// TIA Portal V17 export
// export: Created 2025-08-05T09:35:57.6788297Z, ExportSetting WithDefaults, DisplayName Totally Integrated Automation Portal, DisplayVersion V17, DisplayName TIA Portal Openness, DisplayVersion V17, DisplayName TIA Portal Version Control Interface, DisplayVersion V17, DisplayName SINAMICS Startdrive Advanced, DisplayVersion V17, DisplayName SINAMICS Startdrive G130, G150, S120, S150, SINAMICS MV, S210, DisplayVersion V17, DisplayName SINAMICS Startdrive G110M, G120, G120C, G120D, G120P, G115D, DisplayVersion V17, DisplayName STEP 7 Professional, DisplayVersion V17, DisplayName STEP 7 Safety, DisplayVersion V17, DisplayName WinCC Advanced, DisplayVersion V17
FUNCTION_BLOCK "IPG_Weld_Interface"   // FB304, LAD
TITLE = IPG Communication Handling / IPG Weld Interface
{ S7_Optimized_Access := 'FALSE' }
VERSION : 1.0
// stored: AutoNumber true, IsIECCheckEnabled false, SetENOAutomatically false, UDAEnableTagReadback false
   VAR_INPUT
      iScanner : "Scanner_Inputs";
      iYLS : "YLS_Inputs";
      iInstance_Index : Int;
      iYLR_Power_On : Bool;
      bYLR : Bool;
      bYLS : Bool;
   END_VAR
   VAR_OUTPUT
      oScanner : "Scanner_Outputs";
      oYLS : "YLS_Outputs";
      oYLR_Laser_On : Bool;
      oYLR_Reset : Bool;
   END_VAR
   VAR DB_SPECIFIC
      sStep : Int;
      sLast_Step : Int;
      sScanner_Idle : Bool;
      sScanner_Active : Bool;
      sScanner_Error : Bool;
      sScanner_Waiting_Enable : Bool;
      sScanner_Waiting_Strobe : Bool;
      sScanner_Waiting_Start : Bool;
      tJob_Start_ONS { ExternalAccessible := 'False'; ExternalVisible := 'False'; ExternalWritable := 'False'} : Bool;
      tJob_Stop_ONS { ExternalAccessible := 'False'; ExternalVisible := 'False'; ExternalWritable := 'False'} : Bool;
      siScanner_Job : Byte;
      siScanner_Group : Byte;
      soScanner_Job : Byte;
      soScanner_Group : Byte;
      sVersion { S7_SetPoint := 'True'} : Real;
      sStepTimeout : IEC_TIMER;
      sReset_Timer { S7_SetPoint := 'True'} : IEC_TIMER;
      sLog : Array[0..50] of Struct
         Load_Start_Time : Date_And_Time;
         Load_Stop_Time : Date_And_Time;
         Fire_Start_Time : Date_And_Time;
         Fire_Stop_Time : Date_And_Time;
         Job_ID : Byte;
         Group_ID : Byte;
      END_STRUCT;
      sBlankLog : Struct
         Load_Start_Time : Date_And_Time;
         Load_Stop_Time : Date_And_Time;
         Fire_Start_Time : Date_And_Time;
         Fire_Stop_Time : Date_And_Time;
         Job_ID : Byte;
         Group_ID : Byte;
      END_STRUCT;
   END_VAR
   VAR_TEMP
      tLasRes : Bool;
      tStep_Changed_ONS : Bool;
      tPointer : Int;
      tStart_Load_Int : Int;
      tStop_Load_Int : Int;
      tStart_Fire_Int : Int;
      tStop_Fire_Int : Int;
   END_VAR
   VAR_TEMP   // added for the SCL form of the ladder/FBD networks
      _w1 : Bool;
      _w2 : Bool;
   END_VAR
BEGIN

REGION Network 1: Version
   // V1.1
   // Mapped all Scanner and YLS Inputs and Outputs
   // V1.2
   // Added YLR Faults and Interface (need to add condition for Power On of YLR)
   // V2
   // Laser Comm DB Reorder, remove redunudant logic
   // Added Job and Group Log
   // Removed Guide Beam On Fault. Soace reserved.
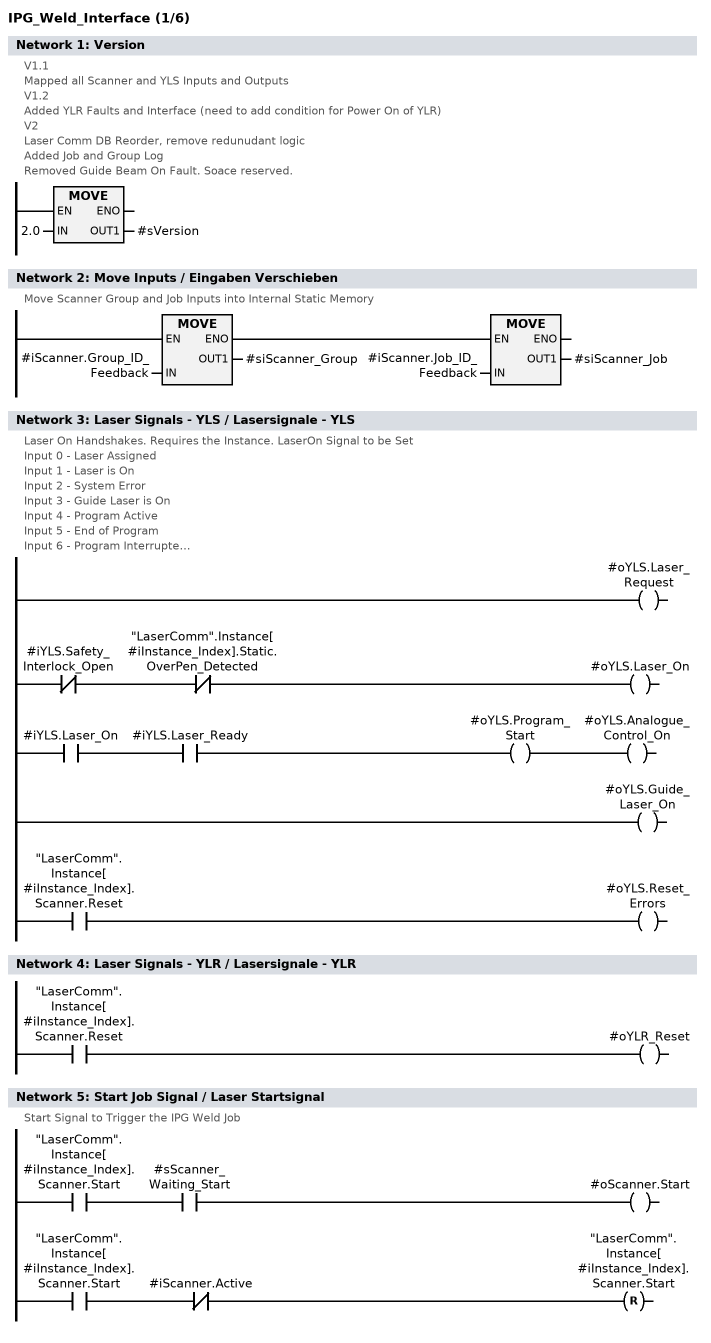
   RUNG wire#powerrail
      Move(in := 2.0, out1 => #sVersion)
   END_RUNG
   // the same network as SCL:
   #sVersion := 2.0;
END_REGION

REGION Network 2: Move Inputs / Eingaben Verschieben
   // Move Scanner Group and Job Inputs into Internal Static Memory
   RUNG wire#powerrail
      Move(in := #iScanner.Group_ID_Feedback, out1 => #siScanner_Group)
      Move(in := #iScanner.Job_ID_Feedback, out1 => #siScanner_Job)
   END_RUNG
   // the same network as SCL:
   #siScanner_Group := #iScanner.Group_ID_Feedback;
   #siScanner_Job := #iScanner.Job_ID_Feedback;
END_REGION

REGION Network 3: Laser Signals - YLS / Lasersignale - YLS
   // Laser On Handshakes. Requires the Instance. LaserOn Signal to be Set
   // Input 0 - Laser Assigned
   // Input 1 - Laser is On
   // Input 2 - System Error
   // Input 3 - Guide Laser is On
   // Input 4 - Program Active
   // Input 5 - End of Program
   // Input 6 - Program Interrupted
   // Input 7 - Analogue Control is On
   // Input 8 - System Warning
   // Input 9 - Laser Ready
   // Input 10 - Emission On
   // 
   // Output 0 - Laser Request (should always be On)
   // Output 1 - Laser On
   // Output 2 - Reset Errors
   // Output 3 - Guide Laser On
   // Output 4 - Program Start
   // Output 5 - Program Stop
   // Output 6 - Reserved
   // Output 7 - Analogue Control On
   RUNG wire#powerrail
      Coil( #oYLS.Laser_Request )
   END_RUNG
   RUNG wire#powerrail
      I_Contact( #iYLS.Safety_Interlock_Open )
      I_Contact( "LaserComm".Instance[#iInstance_Index].Static.OverPen_Detected )
      Coil( #oYLS.Laser_On )
   END_RUNG
   RUNG wire#powerrail
      Contact( #iYLS.Laser_On )
      Contact( #iYLS.Laser_Ready )
      Coil( #oYLS.Program_Start )
      Coil( #oYLS.Analogue_Control_On )
   END_RUNG
   RUNG wire#powerrail
      Coil( #oYLS.Guide_Laser_On )
   END_RUNG
   RUNG wire#powerrail
      Contact( "LaserComm".Instance[#iInstance_Index].Scanner.Reset )
      Coil( #oYLS.Reset_Errors )
   END_RUNG
   // the same network as SCL:
   #oYLS.Laser_Request := TRUE;
   #oYLS.Laser_On := NOT #iYLS.Safety_Interlock_Open AND NOT "LaserComm".Instance[#iInstance_Index].Static.OverPen_Detected;
   #oYLS.Program_Start := #iYLS.Laser_On AND #iYLS.Laser_Ready;
   #oYLS.Analogue_Control_On := #oYLS.Program_Start;
   #oYLS.Guide_Laser_On := TRUE;
   #oYLS.Reset_Errors := "LaserComm".Instance[#iInstance_Index].Scanner.Reset;
END_REGION

REGION Network 4: Laser Signals - YLR / Lasersignale - YLR
   RUNG wire#powerrail
      Contact( "LaserComm".Instance[#iInstance_Index].Scanner.Reset )
      Coil( #oYLR_Reset )
   END_RUNG
   // the same network as SCL:
   #oYLR_Reset := "LaserComm".Instance[#iInstance_Index].Scanner.Reset;
END_REGION

REGION Network 5: Start Job Signal / Laser Startsignal
   // Start Signal to Trigger the IPG Weld Job
   RUNG wire#powerrail
      Contact( "LaserComm".Instance[#iInstance_Index].Scanner.Start )
      Contact( #sScanner_Waiting_Start )
      Coil( #oScanner.Start )
   END_RUNG
   RUNG wire#powerrail
      Contact( "LaserComm".Instance[#iInstance_Index].Scanner.Start )
      I_Contact( #iScanner.Active )
      R_Coil( "LaserComm".Instance[#iInstance_Index].Scanner.Start )
   END_RUNG
   // the same network as SCL:
   #oScanner.Start := "LaserComm".Instance[#iInstance_Index].Scanner.Start AND #sScanner_Waiting_Start;
   IF "LaserComm".Instance[#iInstance_Index].Scanner.Start AND NOT #iScanner.Active THEN
       "LaserComm".Instance[#iInstance_Index].Scanner.Start := FALSE;
   END_IF;
END_REGION

REGION Network 6: Log Fire Time Handling
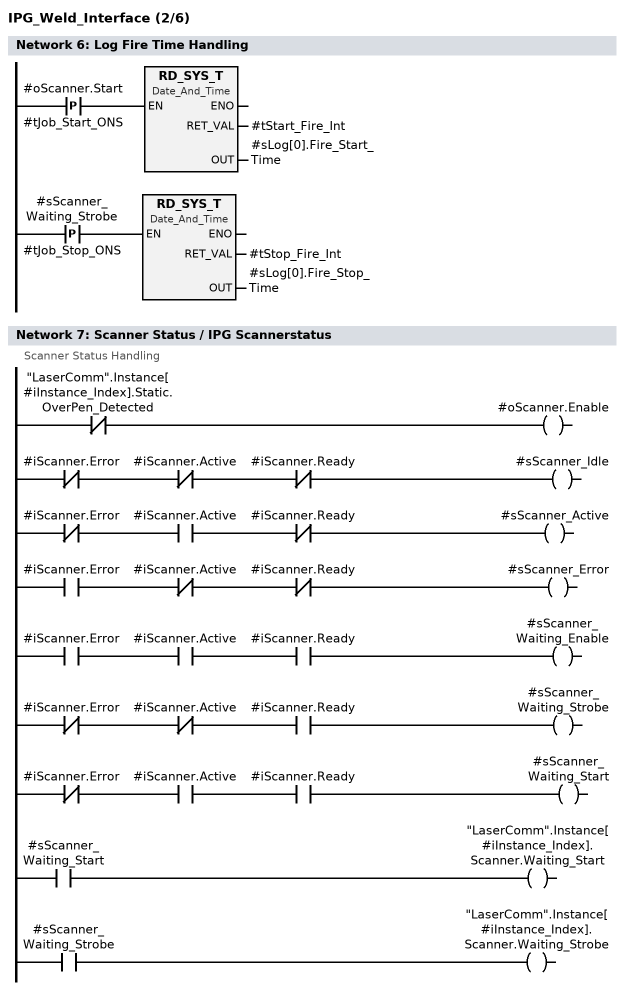
   RUNG wire#powerrail
      P_Contact(operand := #oScanner.Start, bit := #tJob_Start_ONS)
      { S7_Templates := "date_type := Date_And_Time" } RD_SYS_T(RET_VAL => #tStart_Fire_Int, OUT => #sLog[0].Fire_Start_Time)
   END_RUNG
   RUNG wire#powerrail
      P_Contact(operand := #sScanner_Waiting_Strobe, bit := #tJob_Stop_ONS)
      { S7_Templates := "date_type := Date_And_Time" } RD_SYS_T(RET_VAL => #tStop_Fire_Int, OUT => #sLog[0].Fire_Stop_Time)
   END_RUNG
   // the same network as SCL:
   #_w1 := #oScanner.Start AND NOT #tJob_Start_ONS;   // rising edge of #oScanner.Start
   #tJob_Start_ONS := #oScanner.Start;
   IF #_w1 THEN #tStart_Fire_Int := RD_SYS_T(OUT => #sLog[0].Fire_Start_Time); END_IF;
   #_w2 := #sScanner_Waiting_Strobe AND NOT #tJob_Stop_ONS;   // rising edge of #sScanner_Waiting_Strobe
   #tJob_Stop_ONS := #sScanner_Waiting_Strobe;
   IF #_w2 THEN #tStop_Fire_Int := RD_SYS_T(OUT => #sLog[0].Fire_Stop_Time); END_IF;
END_REGION

REGION Network 7: Scanner Status / IPG Scannerstatus
   // Scanner Status Handling
   RUNG wire#powerrail
      I_Contact( "LaserComm".Instance[#iInstance_Index].Static.OverPen_Detected )
      Coil( #oScanner.Enable )
   END_RUNG
   RUNG wire#powerrail
      I_Contact( #iScanner.Error )
      I_Contact( #iScanner.Active )
      I_Contact( #iScanner.Ready )
      Coil( #sScanner_Idle )
   END_RUNG
   RUNG wire#powerrail
      I_Contact( #iScanner.Error )
      Contact( #iScanner.Active )
      I_Contact( #iScanner.Ready )
      Coil( #sScanner_Active )
   END_RUNG
   RUNG wire#powerrail
      Contact( #iScanner.Error )
      I_Contact( #iScanner.Active )
      I_Contact( #iScanner.Ready )
      Coil( #sScanner_Error )
   END_RUNG
   RUNG wire#powerrail
      Contact( #iScanner.Error )
      Contact( #iScanner.Active )
      Contact( #iScanner.Ready )
      Coil( #sScanner_Waiting_Enable )
   END_RUNG
   RUNG wire#powerrail
      I_Contact( #iScanner.Error )
      I_Contact( #iScanner.Active )
      Contact( #iScanner.Ready )
      Coil( #sScanner_Waiting_Strobe )
   END_RUNG
   RUNG wire#powerrail
      I_Contact( #iScanner.Error )
      Contact( #iScanner.Active )
      Contact( #iScanner.Ready )
      Coil( #sScanner_Waiting_Start )
   END_RUNG
   RUNG wire#powerrail
      Contact( #sScanner_Waiting_Start )
      Coil( "LaserComm".Instance[#iInstance_Index].Scanner.Waiting_Start )
   END_RUNG
   RUNG wire#powerrail
      Contact( #sScanner_Waiting_Strobe )
      Coil( "LaserComm".Instance[#iInstance_Index].Scanner.Waiting_Strobe )
   END_RUNG
   // the same network as SCL:
   #oScanner.Enable := NOT "LaserComm".Instance[#iInstance_Index].Static.OverPen_Detected;
   #sScanner_Idle := NOT #iScanner.Error AND NOT #iScanner.Active AND NOT #iScanner.Ready;
   #sScanner_Active := NOT #iScanner.Error AND #iScanner.Active AND NOT #iScanner.Ready;
   #sScanner_Error := #iScanner.Error AND NOT #iScanner.Active AND NOT #iScanner.Ready;
   #sScanner_Waiting_Enable := #iScanner.Error AND #iScanner.Active AND #iScanner.Ready;
   #sScanner_Waiting_Strobe := NOT #iScanner.Error AND NOT #iScanner.Active AND #iScanner.Ready;
   #sScanner_Waiting_Start := NOT #iScanner.Error AND #iScanner.Active AND #iScanner.Ready;
   "LaserComm".Instance[#iInstance_Index].Scanner.Waiting_Start := #sScanner_Waiting_Start;
   "LaserComm".Instance[#iInstance_Index].Scanner.Waiting_Strobe := #sScanner_Waiting_Strobe;
END_REGION

REGION Network 8: Step 0 / Schritt 0
   // Initial Step. Wait for Scanner Ready to Begin with Job and Group Not 0. / Job und Gruppen ID Laden
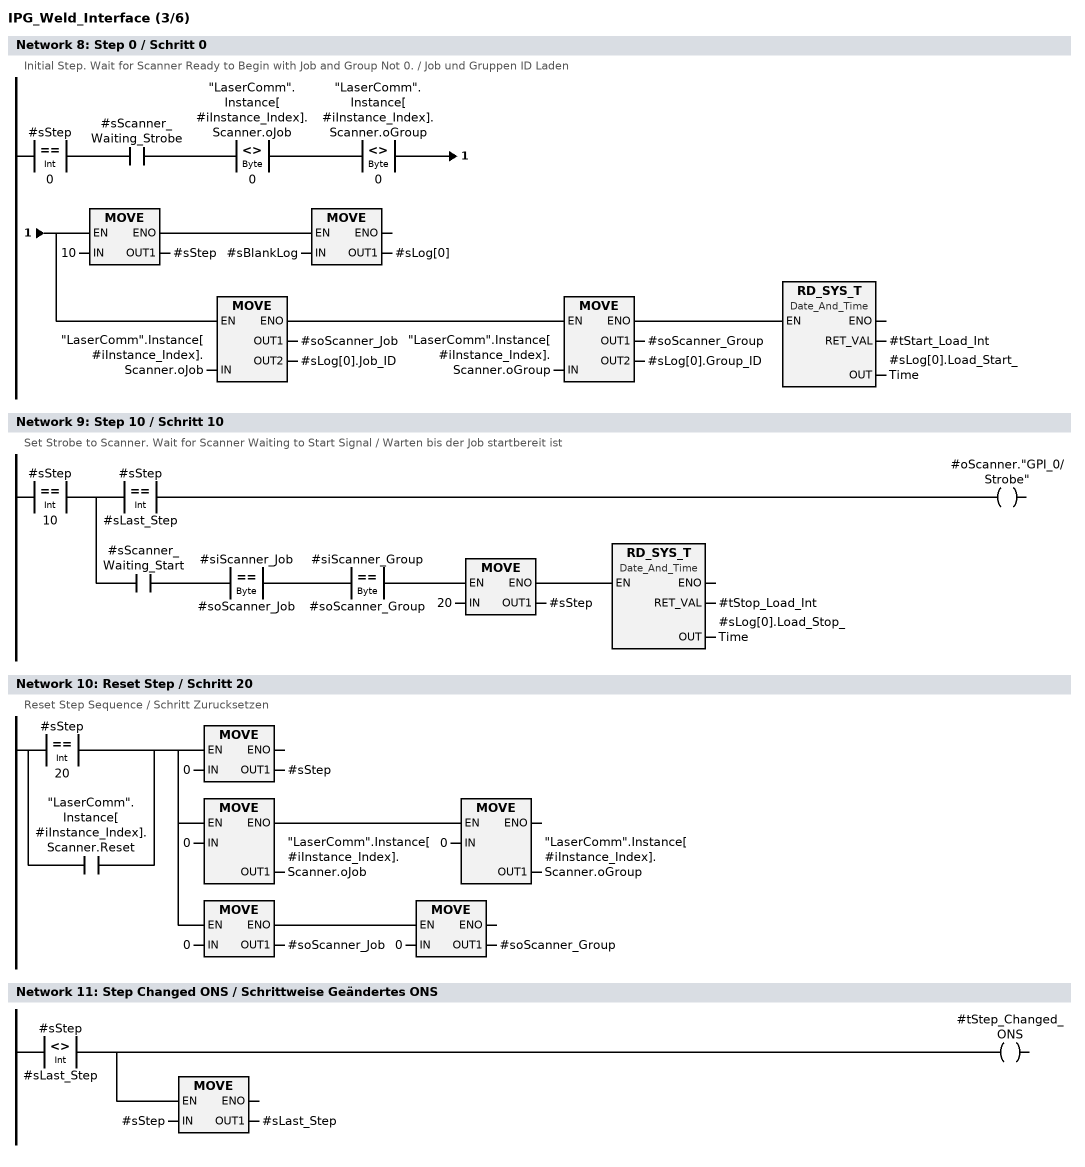
   RUNG wire#powerrail
      { S7_Templates := "SrcType := Int" } EQ_Contact(in1 := #sStep, in2 := 0)
      Contact( #sScanner_Waiting_Strobe )
      { S7_Templates := "SrcType := Byte" } NE_Contact(in1 := "LaserComm".Instance[#iInstance_Index].Scanner.oJob, in2 := 0)
      { S7_Templates := "SrcType := Byte" } NE_Contact(in1 := "LaserComm".Instance[#iInstance_Index].Scanner.oGroup, in2 := 0)
      wire#w1
      Move(in := 10, out1 => #sStep)
      Move(in := #sBlankLog, out1 => #sLog[0])
   END_RUNG
   RUNG wire#w1
      Move(in := "LaserComm".Instance[#iInstance_Index].Scanner.oJob, out1 => #soScanner_Job, out2 => #sLog[0].Job_ID)
      Move(in := "LaserComm".Instance[#iInstance_Index].Scanner.oGroup, out1 => #soScanner_Group, out2 => #sLog[0].Group_ID)
      { S7_Templates := "date_type := Date_And_Time" } RD_SYS_T(RET_VAL => #tStart_Load_Int, OUT => #sLog[0].Load_Start_Time)
   END_RUNG
   // the same network as SCL:
   #_w1 := (#sStep = 0) AND #sScanner_Waiting_Strobe AND ("LaserComm".Instance[#iInstance_Index].Scanner.oJob <> 0) AND ("LaserComm".Instance[#iInstance_Index].Scanner.oGroup <> 0);
   #_w2 := (#sStep = 0) AND #sScanner_Waiting_Strobe AND ("LaserComm".Instance[#iInstance_Index].Scanner.oJob <> 0) AND ("LaserComm".Instance[#iInstance_Index].Scanner.oGroup <> 0);
   IF #_w2 THEN
       #sStep := 10;
       #sLog[0] := #sBlankLog;
   END_IF;
   IF #_w1 THEN
       #soScanner_Job := "LaserComm".Instance[#iInstance_Index].Scanner.oJob;
       #sLog[0].Job_ID := "LaserComm".Instance[#iInstance_Index].Scanner.oJob;
       #soScanner_Group := "LaserComm".Instance[#iInstance_Index].Scanner.oGroup;
       #sLog[0].Group_ID := "LaserComm".Instance[#iInstance_Index].Scanner.oGroup;
       #tStart_Load_Int := RD_SYS_T(OUT => #sLog[0].Load_Start_Time);
   END_IF;
END_REGION

REGION Network 9: Step 10 / Schritt 10
   // Set Strobe to Scanner. Wait for Scanner Waiting to Start Signal / Warten bis der Job startbereit ist
   RUNG wire#powerrail
      { S7_Templates := "SrcType := Int" } EQ_Contact(in1 := #sStep, in2 := 10)
      wire#w1
      { S7_Templates := "SrcType := Int" } EQ_Contact(in1 := #sStep, in2 := #sLast_Step)
      Coil( #oScanner."GPI_0/Strobe" )
   END_RUNG
   RUNG wire#w1
      Contact( #sScanner_Waiting_Start )
      { S7_Templates := "SrcType := Byte" } EQ_Contact(in1 := #siScanner_Job, in2 := #soScanner_Job)
      { S7_Templates := "SrcType := Byte" } EQ_Contact(in1 := #siScanner_Group, in2 := #soScanner_Group)
      Move(in := 20, out1 => #sStep)
      { S7_Templates := "date_type := Date_And_Time" } RD_SYS_T(RET_VAL => #tStop_Load_Int, OUT => #sLog[0].Load_Stop_Time)
   END_RUNG
   // the same network as SCL:
   #_w1 := #sStep = 10;
   #oScanner."GPI_0/Strobe" := #_w1 AND (#sStep = #sLast_Step);
   IF #_w1 AND #sScanner_Waiting_Start AND (#siScanner_Job = #soScanner_Job) AND (#siScanner_Group = #soScanner_Group) THEN
       #sStep := 20;
       #tStop_Load_Int := RD_SYS_T(OUT => #sLog[0].Load_Stop_Time);
   END_IF;
END_REGION

REGION Network 10: Reset Step / Schritt 20
   // Reset Step Sequence / Schritt Zurucksetzen
   RUNG wire#powerrail
      { S7_Templates := "SrcType := Int" } EQ_Contact(in1 := #sStep, in2 := 20)
      wire#w1
      Move(in := 0, out1 => #sStep)
   END_RUNG
   RUNG wire#powerrail
      Contact( "LaserComm".Instance[#iInstance_Index].Scanner.Reset )
   END_RUNG wire#w1
   RUNG wire#w1
      Move(in := 0, out1 => "LaserComm".Instance[#iInstance_Index].Scanner.oJob)
      Move(in := 0, out1 => "LaserComm".Instance[#iInstance_Index].Scanner.oGroup)
   END_RUNG
   RUNG wire#w1
      Move(in := 0, out1 => #soScanner_Job)
      Move(in := 0, out1 => #soScanner_Group)
   END_RUNG
   // the same network as SCL:
   #_w1 := (#sStep = 20) OR "LaserComm".Instance[#iInstance_Index].Scanner.Reset;
   IF #_w1 THEN
       #sStep := 0;
       "LaserComm".Instance[#iInstance_Index].Scanner.oJob := 0;
       "LaserComm".Instance[#iInstance_Index].Scanner.oGroup := 0;
       #soScanner_Job := 0;
       #soScanner_Group := 0;
   END_IF;
END_REGION

REGION Network 11: Step Changed ONS / Schrittweise Geändertes ONS
   RUNG wire#powerrail
      { S7_Templates := "SrcType := Int" } NE_Contact(in1 := #sStep, in2 := #sLast_Step)
      wire#w1
      Coil( #tStep_Changed_ONS )
   END_RUNG
   RUNG wire#w1
      { S7_GenerateENO := "TRUE" } Move(in := #sStep, out1 => #sLast_Step)
   END_RUNG
   // the same network as SCL:
   #tStep_Changed_ONS := #sStep <> #sLast_Step;
   IF #tStep_Changed_ONS THEN #sLast_Step := #sStep; END_IF;
END_REGION

REGION Network 12: Reset Flag / Reset Flag Entrigein
   // Clear Reset Flag - Timer Required as Laser Source requires a duration pulse to reset
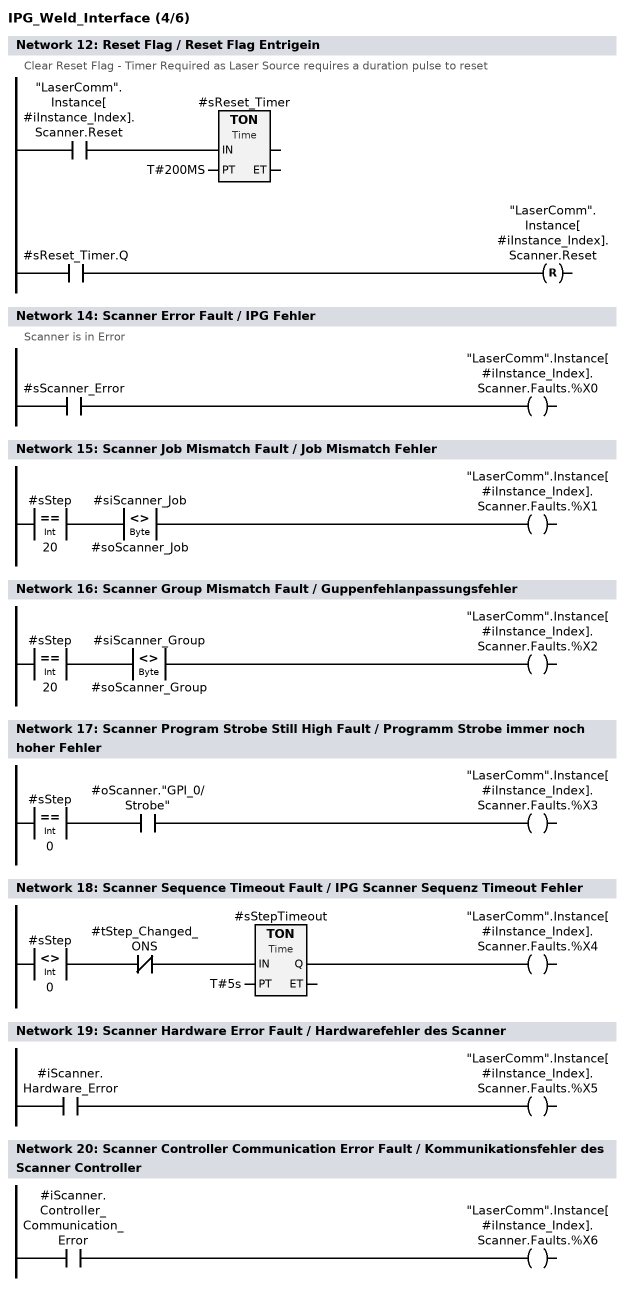
   RUNG wire#powerrail
      Contact( "LaserComm".Instance[#iInstance_Index].Scanner.Reset )
      { S7_Templates := "time_type := Time" } #sReset_Timer.TON(pt := T#200MS, et =>)
   END_RUNG
   RUNG wire#powerrail
      Contact( #sReset_Timer.Q )
      R_Coil( "LaserComm".Instance[#iInstance_Index].Scanner.Reset )
   END_RUNG
   // the same network as SCL:
   #sReset_Timer.TON(IN := "LaserComm".Instance[#iInstance_Index].Scanner.Reset, PT := T#200MS);
   IF #sReset_Timer.Q THEN "LaserComm".Instance[#iInstance_Index].Scanner.Reset := FALSE; END_IF;
END_REGION

REGION Network 13 (SCL): Job Log Handler
   // Records when the last job and group was loaded and fired
   // Job Log Handler

   IF #sLog[0].Job_ID <> 0 AND #sLog[0].Group_ID <> 0 AND #sLog[0].Fire_Stop_Time <> DT#1990-01-01-00:00:00 THEN
       FOR #tPointer := 49 TO 0 BY -1 DO
           #sLog[#tPointer + 1] := #sLog[#tPointer];
       END_FOR;

       #sLog[0] := #sBlankLog;

   END_IF;
END_REGION

REGION Network 14: Scanner Error Fault / IPG Fehler
   // Scanner is in Error
   RUNG wire#powerrail
      Contact( #sScanner_Error )
      Coil( "LaserComm".Instance[#iInstance_Index].Scanner.Faults.%X0 )
   END_RUNG
   // the same network as SCL:
   "LaserComm".Instance[#iInstance_Index].Scanner.Faults.%X0 := #sScanner_Error;
END_REGION

REGION Network 15: Scanner Job Mismatch Fault / Job Mismatch Fehler
   RUNG wire#powerrail
      { S7_Templates := "SrcType := Int" } EQ_Contact(in1 := #sStep, in2 := 20)
      { S7_Templates := "SrcType := Byte" } NE_Contact(in1 := #siScanner_Job, in2 := #soScanner_Job)
      Coil( "LaserComm".Instance[#iInstance_Index].Scanner.Faults.%X1 )
   END_RUNG
   // the same network as SCL:
   "LaserComm".Instance[#iInstance_Index].Scanner.Faults.%X1 := (#sStep = 20) AND (#siScanner_Job <> #soScanner_Job);
END_REGION

REGION Network 16: Scanner Group Mismatch Fault / Guppenfehlanpassungsfehler
   RUNG wire#powerrail
      { S7_Templates := "SrcType := Int" } EQ_Contact(in1 := #sStep, in2 := 20)
      { S7_Templates := "SrcType := Byte" } NE_Contact(in1 := #siScanner_Group, in2 := #soScanner_Group)
      Coil( "LaserComm".Instance[#iInstance_Index].Scanner.Faults.%X2 )
   END_RUNG
   // the same network as SCL:
   "LaserComm".Instance[#iInstance_Index].Scanner.Faults.%X2 := (#sStep = 20) AND (#siScanner_Group <> #soScanner_Group);
END_REGION

REGION Network 17: Scanner Program Strobe Still High Fault / Programm Strobe immer noch hoher Fehler
   RUNG wire#powerrail
      { S7_Templates := "SrcType := Int" } EQ_Contact(in1 := #sStep, in2 := 0)
      Contact( #oScanner."GPI_0/Strobe" )
      Coil( "LaserComm".Instance[#iInstance_Index].Scanner.Faults.%X3 )
   END_RUNG
   // the same network as SCL:
   "LaserComm".Instance[#iInstance_Index].Scanner.Faults.%X3 := (#sStep = 0) AND #oScanner."GPI_0/Strobe";
END_REGION

REGION Network 18: Scanner Sequence Timeout Fault / IPG Scanner Sequenz Timeout Fehler
   RUNG wire#powerrail
      { S7_Templates := "SrcType := Int" } NE_Contact(in1 := #sStep, in2 := 0)
      I_Contact( #tStep_Changed_ONS )
      { S7_Templates := "time_type := Time" } #sStepTimeout.TON(pt := T#5s, et =>)
      Coil( "LaserComm".Instance[#iInstance_Index].Scanner.Faults.%X4 )
   END_RUNG
   // the same network as SCL:
   #sStepTimeout.TON(IN := (#sStep <> 0) AND NOT #tStep_Changed_ONS, PT := T#5s);
   "LaserComm".Instance[#iInstance_Index].Scanner.Faults.%X4 := #sStepTimeout.Q;
END_REGION

REGION Network 19: Scanner Hardware Error Fault / Hardwarefehler des Scanner
   RUNG wire#powerrail
      Contact( #iScanner.Hardware_Error )
      Coil( "LaserComm".Instance[#iInstance_Index].Scanner.Faults.%X5 )
   END_RUNG
   // the same network as SCL:
   "LaserComm".Instance[#iInstance_Index].Scanner.Faults.%X5 := #iScanner.Hardware_Error;
END_REGION

REGION Network 20: Scanner Controller Communication Error Fault / Kommunikationsfehler des Scanner Controller
   RUNG wire#powerrail
      Contact( #iScanner.Controller_Communication_Error )
      Coil( "LaserComm".Instance[#iInstance_Index].Scanner.Faults.%X6 )
   END_RUNG
   // the same network as SCL:
   "LaserComm".Instance[#iInstance_Index].Scanner.Faults.%X6 := #iScanner.Controller_Communication_Error;
END_REGION

REGION Network 21: Scanner Head Communication Error Fault / Fehler bei derKommunikation mit dem Scannerkopf
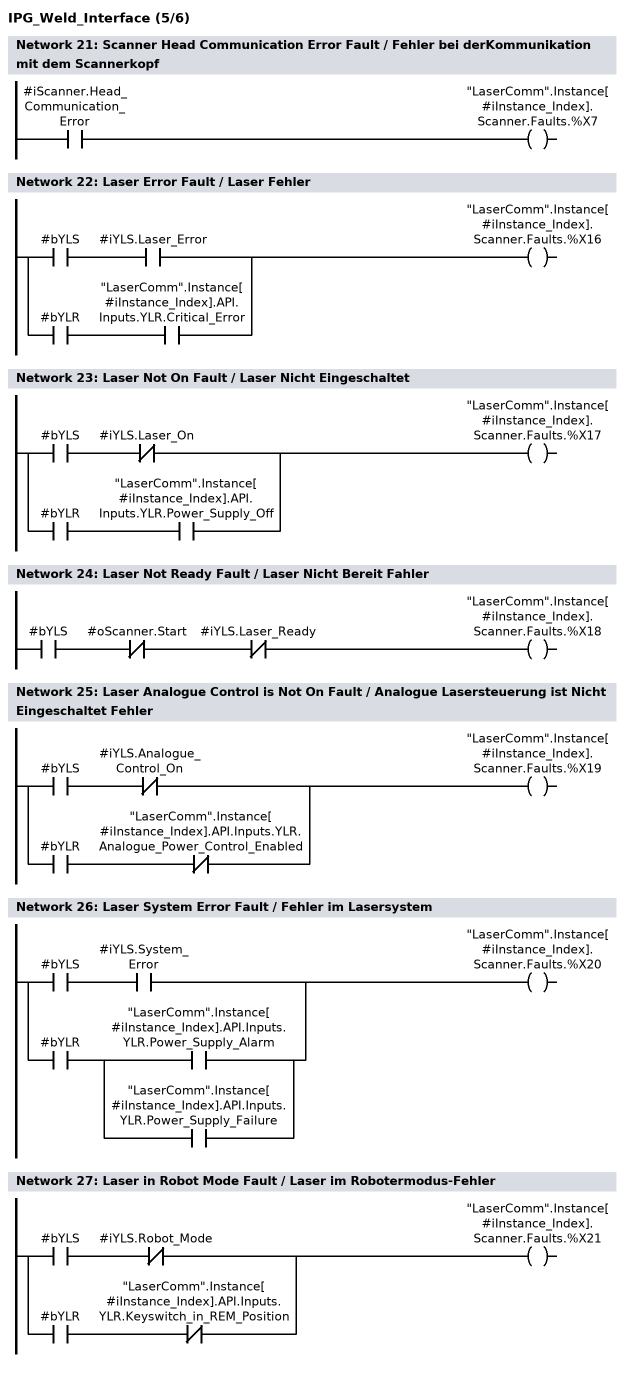
   RUNG wire#powerrail
      Contact( #iScanner.Head_Communication_Error )
      Coil( "LaserComm".Instance[#iInstance_Index].Scanner.Faults.%X7 )
   END_RUNG
   // the same network as SCL:
   "LaserComm".Instance[#iInstance_Index].Scanner.Faults.%X7 := #iScanner.Head_Communication_Error;
END_REGION

REGION Network 22: Laser Error Fault / Laser Fehler
   RUNG wire#powerrail
      Contact( #bYLS )
      Contact( #iYLS.Laser_Error )
      wire#w1
      Coil( "LaserComm".Instance[#iInstance_Index].Scanner.Faults.%X16 )
   END_RUNG
   RUNG wire#powerrail
      Contact( #bYLR )
      Contact( "LaserComm".Instance[#iInstance_Index].API.Inputs.YLR.Critical_Error )
   END_RUNG wire#w1
   // the same network as SCL:
   "LaserComm".Instance[#iInstance_Index].Scanner.Faults.%X16 := (#bYLS AND #iYLS.Laser_Error) OR (#bYLR AND "LaserComm".Instance[#iInstance_Index].API.Inputs.YLR.Critical_Error);
END_REGION

REGION Network 23: Laser Not On Fault / Laser Nicht Eingeschaltet
   RUNG wire#powerrail
      Contact( #bYLS )
      I_Contact( #iYLS.Laser_On )
      wire#w1
      Coil( "LaserComm".Instance[#iInstance_Index].Scanner.Faults.%X17 )
   END_RUNG
   RUNG wire#powerrail
      Contact( #bYLR )
      Contact( "LaserComm".Instance[#iInstance_Index].API.Inputs.YLR.Power_Supply_Off )
   END_RUNG wire#w1
   // the same network as SCL:
   "LaserComm".Instance[#iInstance_Index].Scanner.Faults.%X17 := (#bYLS AND NOT #iYLS.Laser_On) OR (#bYLR AND "LaserComm".Instance[#iInstance_Index].API.Inputs.YLR.Power_Supply_Off);
END_REGION

REGION Network 24: Laser Not Ready Fault / Laser Nicht Bereit Fahler
   RUNG wire#powerrail
      Contact( #bYLS )
      I_Contact( #oScanner.Start )
      I_Contact( #iYLS.Laser_Ready )
      Coil( "LaserComm".Instance[#iInstance_Index].Scanner.Faults.%X18 )
   END_RUNG
   // the same network as SCL:
   "LaserComm".Instance[#iInstance_Index].Scanner.Faults.%X18 := #bYLS AND NOT #oScanner.Start AND NOT #iYLS.Laser_Ready;
END_REGION

REGION Network 25: Laser Analogue Control is Not On Fault / Analogue Lasersteuerung ist Nicht Eingeschaltet Fehler
   RUNG wire#powerrail
      Contact( #bYLS )
      I_Contact( #iYLS.Analogue_Control_On )
      wire#w1
      Coil( "LaserComm".Instance[#iInstance_Index].Scanner.Faults.%X19 )
   END_RUNG
   RUNG wire#powerrail
      Contact( #bYLR )
      I_Contact( "LaserComm".Instance[#iInstance_Index].API.Inputs.YLR.Analogue_Power_Control_Enabled )
   END_RUNG wire#w1
   // the same network as SCL:
   "LaserComm".Instance[#iInstance_Index].Scanner.Faults.%X19 := (#bYLS AND NOT #iYLS.Analogue_Control_On) OR (#bYLR AND NOT "LaserComm".Instance[#iInstance_Index].API.Inputs.YLR.Analogue_Power_Control_Enabled);
END_REGION

REGION Network 26: Laser System Error Fault / Fehler im Lasersystem
   RUNG wire#powerrail
      Contact( #bYLS )
      Contact( #iYLS.System_Error )
      wire#w1
      Coil( "LaserComm".Instance[#iInstance_Index].Scanner.Faults.%X20 )
   END_RUNG
   RUNG wire#powerrail
      Contact( #bYLR )
      wire#w2
      Contact( "LaserComm".Instance[#iInstance_Index].API.Inputs.YLR.Power_Supply_Alarm )
   END_RUNG wire#w1
   RUNG wire#w2
      Contact( "LaserComm".Instance[#iInstance_Index].API.Inputs.YLR.Power_Supply_Failure )
   END_RUNG wire#w1
   // the same network as SCL:
   "LaserComm".Instance[#iInstance_Index].Scanner.Faults.%X20 := (#bYLS AND #iYLS.System_Error) OR (#bYLR AND ("LaserComm".Instance[#iInstance_Index].API.Inputs.YLR.Power_Supply_Alarm OR "LaserComm".Instance[#iInstance_Index].API.Inputs.YLR.Power_Supply_Failure));
END_REGION

REGION Network 27: Laser in Robot Mode Fault / Laser im Robotermodus-Fehler
   RUNG wire#powerrail
      Contact( #bYLS )
      I_Contact( #iYLS.Robot_Mode )
      wire#w1
      Coil( "LaserComm".Instance[#iInstance_Index].Scanner.Faults.%X21 )
   END_RUNG
   RUNG wire#powerrail
      Contact( #bYLR )
      I_Contact( "LaserComm".Instance[#iInstance_Index].API.Inputs.YLR.Keyswitch_in_REM_Position )
   END_RUNG wire#w1
   // the same network as SCL:
   "LaserComm".Instance[#iInstance_Index].Scanner.Faults.%X21 := (#bYLS AND NOT #iYLS.Robot_Mode) OR (#bYLR AND NOT "LaserComm".Instance[#iInstance_Index].API.Inputs.YLR.Keyswitch_in_REM_Position);
END_REGION

REGION Network 28: Laser Interlock Open Fault / Fehler Laserverriegelung offen
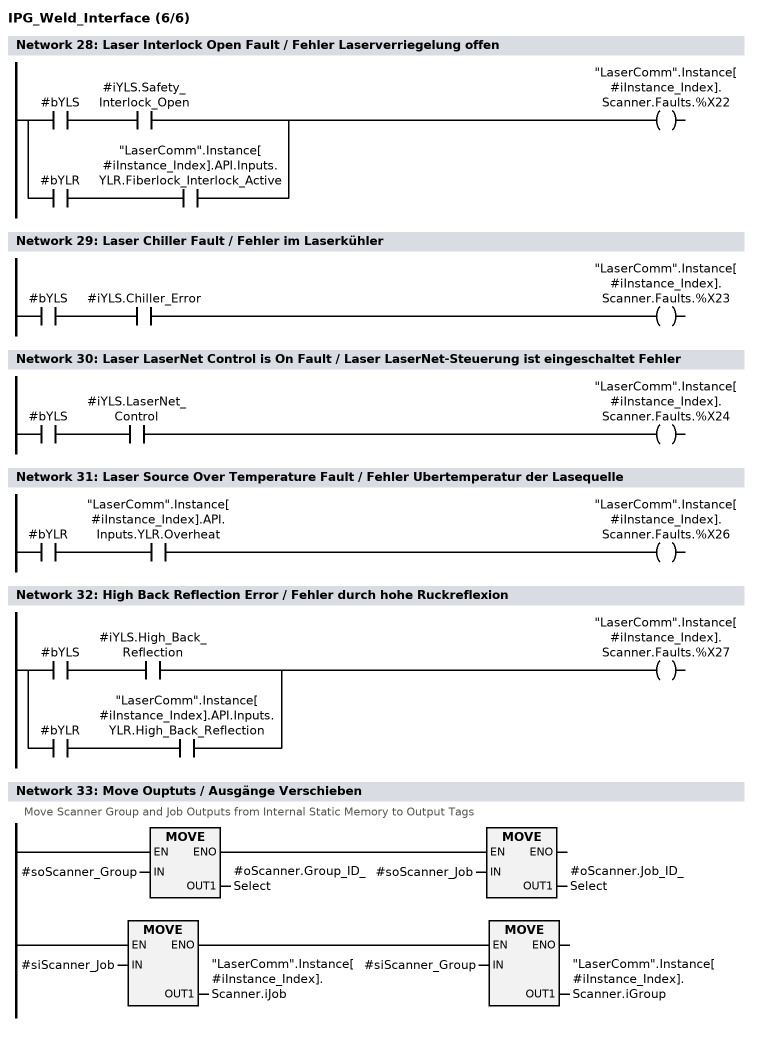
   RUNG wire#powerrail
      Contact( #bYLS )
      Contact( #iYLS.Safety_Interlock_Open )
      wire#w1
      Coil( "LaserComm".Instance[#iInstance_Index].Scanner.Faults.%X22 )
   END_RUNG
   RUNG wire#powerrail
      Contact( #bYLR )
      Contact( "LaserComm".Instance[#iInstance_Index].API.Inputs.YLR.Fiberlock_Interlock_Active )
   END_RUNG wire#w1
   // the same network as SCL:
   "LaserComm".Instance[#iInstance_Index].Scanner.Faults.%X22 := (#bYLS AND #iYLS.Safety_Interlock_Open) OR (#bYLR AND "LaserComm".Instance[#iInstance_Index].API.Inputs.YLR.Fiberlock_Interlock_Active);
END_REGION

REGION Network 29: Laser Chiller Fault / Fehler im Laserkühler
   RUNG wire#powerrail
      Contact( #bYLS )
      Contact( #iYLS.Chiller_Error )
      Coil( "LaserComm".Instance[#iInstance_Index].Scanner.Faults.%X23 )
   END_RUNG
   // the same network as SCL:
   "LaserComm".Instance[#iInstance_Index].Scanner.Faults.%X23 := #bYLS AND #iYLS.Chiller_Error;
END_REGION

REGION Network 30: Laser LaserNet Control is On Fault / Laser LaserNet-Steuerung ist eingeschaltet Fehler
   RUNG wire#powerrail
      Contact( #bYLS )
      Contact( #iYLS.LaserNet_Control )
      Coil( "LaserComm".Instance[#iInstance_Index].Scanner.Faults.%X24 )
   END_RUNG
   // the same network as SCL:
   "LaserComm".Instance[#iInstance_Index].Scanner.Faults.%X24 := #bYLS AND #iYLS.LaserNet_Control;
END_REGION

REGION Network 31: Laser Source Over Temperature Fault / Fehler Ubertemperatur der Lasequelle
   RUNG wire#powerrail
      Contact( #bYLR )
      Contact( "LaserComm".Instance[#iInstance_Index].API.Inputs.YLR.Overheat )
      Coil( "LaserComm".Instance[#iInstance_Index].Scanner.Faults.%X26 )
   END_RUNG
   // the same network as SCL:
   "LaserComm".Instance[#iInstance_Index].Scanner.Faults.%X26 := #bYLR AND "LaserComm".Instance[#iInstance_Index].API.Inputs.YLR.Overheat;
END_REGION

REGION Network 32: High Back Reflection Error / Fehler durch hohe Ruckreflexion
   RUNG wire#powerrail
      Contact( #bYLS )
      Contact( #iYLS.High_Back_Reflection )
      wire#w1
      Coil( "LaserComm".Instance[#iInstance_Index].Scanner.Faults.%X27 )
   END_RUNG
   RUNG wire#powerrail
      Contact( #bYLR )
      Contact( "LaserComm".Instance[#iInstance_Index].API.Inputs.YLR.High_Back_Reflection )
   END_RUNG wire#w1
   // the same network as SCL:
   "LaserComm".Instance[#iInstance_Index].Scanner.Faults.%X27 := (#bYLS AND #iYLS.High_Back_Reflection) OR (#bYLR AND "LaserComm".Instance[#iInstance_Index].API.Inputs.YLR.High_Back_Reflection);
END_REGION

REGION Network 33: Move Ouptuts / Ausgänge Verschieben
   // Move Scanner Group and Job Outputs from Internal Static Memory to Output Tags
   RUNG wire#powerrail
      Move(in := #soScanner_Group, out1 => #oScanner.Group_ID_Select)
      Move(in := #soScanner_Job, out1 => #oScanner.Job_ID_Select)
   END_RUNG
   RUNG wire#powerrail
      Move(in := #siScanner_Job, out1 => "LaserComm".Instance[#iInstance_Index].Scanner.iJob)
      Move(in := #siScanner_Group, out1 => "LaserComm".Instance[#iInstance_Index].Scanner.iGroup)
   END_RUNG
   // the same network as SCL:
   #oScanner.Group_ID_Select := #soScanner_Group;
   #oScanner.Job_ID_Select := #soScanner_Job;
   "LaserComm".Instance[#iInstance_Index].Scanner.iJob := #siScanner_Job;
   "LaserComm".Instance[#iInstance_Index].Scanner.iGroup := #siScanner_Group;
END_REGION
END_FUNCTION_BLOCK
